// TIA Portal V15.1 export
// export: Created 2020-12-23T11:16:33.2864918Z, ExportSetting WithDefaults, WithReadOnly, DisplayName Totally Integrated Automation Portal, DisplayVersion V15.1 Update 3, DisplayName TIA Portal Openness, DisplayVersion V15.1, DisplayName STEP 7 Professional, DisplayVersion V15.1 Update 3, DisplayName WinCC Advanced, DisplayVersion V15.1 Update 3
DATA_BLOCK "DBVALVES"   // DB1330
{ S7_Optimized_Access := 'TRUE' }
VERSION : 0.1
// stored: AutoNumber false, CodeModifiedDate 2020-12-23T11:16:22.2079236Z, CompileDate 2020-12-23T11:16:23.5925798Z, CreationDate 2020-12-23T11:14:57.9258238Z, DBAccessibleFromOPCUA true, DownloadWithoutReinit false, InterfaceModifiedDate 2020-12-23T11:16:22.2079236Z, IsConsistent true, IsKnowHowProtected false, IsOnlyStoredInLoadMemory false, IsPLCDB false, IsRetainMemResEnabled false, IsWriteProtectedInAS false, MemoryReserve 100, ModifiedDate 2020-12-23T11:16:22.2079236Z, ParameterModified 2020-12-23T11:16:22.2079236Z, StructureModified 2020-12-23T11:16:22.2079236Z
BEGIN
END_DATA_BLOCK
